INTERFACE I_Crane

PROPERTY bBusy : BOOL
GET
END_GET
SET
END_SET
END_PROPERTY

PROPERTY bError : BOOL
GET
END_GET
SET
END_SET
END_PROPERTY

PROPERTY eState : E_CraneState
GET
END_GET
SET
END_SET
END_PROPERTY

METHOD M_MoveToPostion : BOOL
VAR_INPUT
	stTarget : ST_Position;
END_VAR
END_METHOD

METHOD M_Pick : BOOL
VAR_INPUT
END_VAR
END_METHOD

METHOD M_Place : BOOL
VAR_INPUT
END_VAR
END_METHOD

METHOD M_Reset : BOOL
VAR_INPUT
END_VAR
END_METHOD

END_INTERFACE

(* stored: Version 1.1.0.1, ProductVersion 3.1.4024.16
   Itf I_Crane: Id {0aaef61f-066b-45f1-a3b6-75f98e8b3795}
   Property bBusy: Id {7a2e4410-aaa1-4e68-8768-d894eb967ba7}
   Get Get: Id {16c0bb63-db0c-4c58-ae8b-ed97f6cf6529}
   Set Set: Id {be85927b-4004-4bce-8257-d2a009dc5c24}
   Property bError: Id {dba9e56a-fa95-4628-91da-91952417a079}
   Get Get: Id {2f446fee-cced-48e9-870d-c06d674ed1e1}
   Set Set: Id {52bc36fd-d084-4d8c-948d-897b2f25555b}
   Property eState: Id {a9bdf396-aa83-4303-b1e4-3394e6e9ec16}
   Get Get: Id {7f733256-00d7-4d73-a94d-be26431832f6}
   Set Set: Id {7e4a826c-d313-4b60-a5c0-57e9c2ce254a}
   Method M_MoveToPostion: Id {0c5d9832-797d-4201-9156-b0ce7022f959}
   Method M_Pick: Id {9e6cf4c1-5f1c-4839-a8c6-1fb522f2cbc7}
   Method M_Place: Id {07225ac2-4374-48d0-8e94-d3310713b1c4}
   Method M_Reset: Id {b2067ad9-ddf1-4741-9e86-70964d6c99b1} *)
